Omron CX-Programmer project NewProject (CX-Programmer 9.73)

# PLC NewPLC1: CP1E N20

## Global symbols (name address type ; comment)
0.01 BOOL  ; SENSOR 1
0.03 BOOL  ; RESET
100.00 BOOL  ; OUTPUT
C001 BOOL  ; PEMBILANG

## Program NewProgram1 (cyclic task 0)

### Section Section1

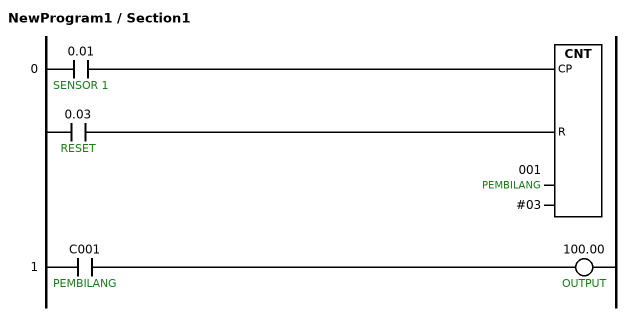
; rung 0
LD 0.01  ; SENSOR 1
LD 0.03  ; RESET
CNT 001 #03  ; PEMBILANG
; rung 1
LD C001  ; PEMBILANG
OUT 100.00  ; OUTPUT

### Section END
; rung 0
END(001)